{attribute 'GeneratedUsingTerminal: EK1122-0000-0018'}
{attribute addProperty BoxType "EK1122-0000-0018"}
{attribute addProperty Id "Beckhoff_EL69xxsub_EK1100EK1100_1FC0878B2"}
{attribute addProperty CRC "3517181034"}
{attribute addProperty Size "2"}
TYPE Beckhoff_EL69xxEK1122_D1A3EC6A EXTENDS EK1122_1FC0878B :
STRUCT
	{attribute addProperty Name "Beckhoff_EL69xxsub_EK1100"}
	{attribute addProperty PreviousPort "Beckhoff EL69xxEK1122 : D"}
	Beckhoff_EL69xxsub_EK1100 : EK1100_1FC0878B;
END_STRUCT
END_TYPE

(* stored: Version 1.2.0.0, ProductVersion 3.1.4024.9
   DUT Beckhoff_EL69xxEK1122_D1A3EC6A: Id {9115c134-04b5-4226-99f7-434dea190040} *)
